//***********************************************************************************
// Concrete Pump
//***********************************************************************************

// concrete pump power control is from pump itself
P_CP1_Enable();
P_CP1_Check(b_set_run := fb_SetOutputDataToIO.b_CP1_Forward_On,
			b_check_mode_on := fb_SetOutputDataToIO.b_CP1_Check_On,
			t_check_duration := fb_setConfig._t_CP1_Check_Duration,
			);


//***********************************************************************************
// Acceleration Pump
//***********************************************************************************

// Acceleration Pump 1 check
P_AP1_Check(b_set_run := fb_SetOutputDataToIO.b_AP1_Run,
			b_check_mode_on := fb_SetOutputDataToIO.b_AP1_Check_On,
			t_check_duration := fb_setConfig._t_AP1_Check_Duration,
			);
// Check for Acceleration Pump 1 state
IF NOT fb_SetOutputDataToIO.b_AP1_Check_On THEN
//
// Acceleration Pump 1 On/Off
	P_AP1_OnOff(b_set_run := fb_SetOutputDataToIO.b_AP1_Run);
END_IF

//***********************************************************************************
// Superplasticizer Pump
//***********************************************************************************

// Superplasticizer Pump 1 Check (220916 WT
P_SP1_Check(b_set_run := fb_SetOutputDataToIO.b_SP1_Run,
			b_check_mode_on := fb_SetOutputDataToIO.b_SP1_Check_On,
			t_check_duration := fb_setConfig._t_SP1_Check_Duration,
			);
IF NOT fb_SetOutputDataToIO.b_SP1_Check_On THEN
	P_SP1_OnOff(b_set_run := fb_SetOutputDataToIO.b_SP1_Run);
END_IF

//***********************************************************************************
// Get out put data from PLC
//***********************************************************************************
fb_getOutputData(
	
	//CC1
	b_mode_manual := GVL_RESD.b_Operate_mode_manual,
	b_mode_laptop := GVL_RESD.b_Operate_mode_laptop, 	
	b_mode_robot := GVL_RESD.b_Operate_mode_robot, 
	b_CC1_power_on := GVL_RESD.b_Concrete_Controller_power_on, 
	n_current_mode := GVL_RESD.n_Concrete_Controller_current_mode,

	//MI1
	b_MI1_Is_Run := GVL_RESD.b_MI1_Is_Run,
	b_MI1_is_ready := GVL_RESD.b_MI1_Is_Ready,
	n_MI1_status_SpeedM1 := GVL_RESD.n_MI1_status_SpeedM1,
	n_MI1_status_SpeedM2 := GVL_RESD.n_MI1_status_SpeedM2,
	f_Status_Torque_Motor_1 := GVL_RESD.f_Status_Torque_Motor_1,
	f_Status_Torque_Motor_2 := GVL_RESD.f_Status_Torque_Motor_2,
	f_MI1_status_temperature_funnel_outlet := GVL_RESD.f_MI1_status_temperature_funnel_outlet, 		
	f_MI1_status_Pressure_funnel_inlet := GVL_RESD.f_MI1_status_Pressure_funnel_inlet, 	
	f_MI1_status_temperature_motor_1  := GVL_RESD.f_MI1_status_temperature_motor_1, 			 
	f_MI1_status_temperature_motor_2  := GVL_RESD.f_MI1_status_temperature_motor_2,

	//CP1
	b_CP1_is_run := GVL_RESD.b_CP1_is_run,
	b_CP1_is_ready := GVL_RESD.b_CP1_is_ready,
	f_CP1_status_temperature_concrete_fresh := GVL_RESD.f_CP1_status_temperature_concrete_fresh,
	f_CP1_status_temperature_Concrete_pump := GVL_RESD.f_CP1_status_temperature_Concrete_pump,
	f_CP1_status_pressure_Concrete_pump := GVL_RESD.f_CP1_status_pressure_Concrete_pump,
	
	//AP1
	b_AP1_is_run := GVL_RESD.b_Admixture_Pump_is_run,
	b_AP1_is_ready := GVL_RESD.b_Admixture_Pump_is_run,
	
	//SP1
	b_SP1_is_run := GVL_RESD.b_Sup_Admixture_Pump_is_run,
	b_SP1_is_ready := GVL_RESD.b_Sup_Admixture_Pump_is_ready,
);

END_PROGRAM

// ---- POUs/Utils/F_Convert_2Byte_to_Int.TcPOU
FUNCTION F_Convert_2Byte_to_Int 

VAR_IN_OUT
	inputNum : INT; 
	dataByte1 : BYTE;
	dataByte2 : BYTE;
END_VAR

VAR
	arrByte : ARRAY [0..1] OF BYTE;
END_VAR

arrByte[0]:= dataByte1;
arrByte[1]:= dataByte2;
MEMCPY(ADR(inputNum), ADR(arrByte), 2);

//F_Convert_Int_to_2Byte:=arrByte;

END_FUNCTION

// ---- POUs/Utils/F_Convert_Byte_to_Bit.TcPOU
FUNCTION  F_Convert_Byte_to_Bit : ARRAY[0..7] OF BOOL
VAR_INPUT
	dataByte : BYTE;
END_VAR

VAR
	arrBool : ARRAY[0..7] OF BOOL;
END_VAR

// ***********************************************************************************
//
// Müller-steinag Gruppe, Kandergrien Einigen, CH-3646 Bern
// ETH Zurich, Building HIF E26, Laura-Hezner-Weg 7, CH-8093 Zürich
// 
// ***********************************************************************************
// 
// PROJECT     :  A061 Digital Casting System 
// FUNCTION    :  Data Converter Byte to Bit
// AUTHOR      :  Weiting Chen
// EMAIL       :  chenw@usi.ch
// Copyright   :  USI Mendrisio; ETH Zürich; Müller-steinag Gruppe (CH) 2023
//
// ***********************************************************************************


// hexadecimal format
arrBool[0] := BYTE_TO_BIT(dataByte AND 16#1);
arrBool[1] := BYTE_TO_BIT(dataByte AND 16#2);
arrBool[2] := BYTE_TO_BIT(dataByte AND 16#4);
arrBool[3] := BYTE_TO_BIT(dataByte AND 16#8);
arrBool[4] := BYTE_TO_BIT(dataByte AND 16#10);
arrBool[5] := BYTE_TO_BIT(dataByte AND 16#20);
arrBool[6] := BYTE_TO_BIT(dataByte AND 16#40);
arrBool[7] := BYTE_TO_BIT(dataByte AND 16#80);

F_Convert_Byte_to_Bit := arrBool;

END_FUNCTION

// ---- POUs/Utils/F_Convert_Int_to_2Byte.TcPOU
FUNCTION F_Convert_Int_to_2Byte
VAR_IN_OUT
	inputNum : INT; 
	dataByte1 : BYTE;
	dataByte2 : BYTE;
END_VAR

VAR
	arrByte : ARRAY [0..1] OF BYTE;
END_VAR

MEMCPY(ADR(arrByte), ADR(inputNum), 2);
dataByte1 := arrByte[0];
dataByte2 := arrByte[1];

//F_Convert_Int_to_2Byte:=arrByte;

END_FUNCTION

// ---- POUs/Utils/F_DecimalData.TcPOU
FUNCTION F_DecimalData : LREAL
VAR_INPUT
	
	f_value_input : REAL;
	// decimal places
	n_decimal_digit : INT;
	// Round or not
	b_round_data: BOOL;

END_VAR
VAR_OUTPUT	
	f_value_output : REAL;
END_VAR
VAR
END_VAR

f_value_output := STRING_TO_REAL(LREAL_TO_FMTSTR(TO_REAL(f_value_input), n_decimal_digit, b_round_data));
F_DecimalData := f_value_output

END_FUNCTION
